// TIA Portal V17 export
// export: Created 2026-04-13T11:12:43.3625871Z, ExportSetting WithDefaults, DisplayName Totally Integrated Automation Portal, DisplayVersion V17 Update 4, DisplayName TIA Portal Openness, DisplayVersion V17 Update 4, DisplayName TIA Portal Version Control Interface, DisplayVersion V17, DisplayName SINAMICS Startdrive Advanced, DisplayVersion V17, DisplayName SINAMICS Startdrive G130, G150, S120, S150, SINAMICS MV, S210, DisplayVersion V17, DisplayName SINAMICS Startdrive G110M, G120, G120C, G120D, G120P, G115D, DisplayVersion V17, DisplayName STEP 7 Professional, DisplayVersion V17 Update 4, DisplayName STEP 7 Safety, DisplayVersion V17, DisplayName WinCC Professional, DisplayVersion V17 Update 4
FUNCTION_BLOCK "1-模拟量输出2"   // FB77, SCL
{ S7_Optimized_Access := 'TRUE' }
VERSION : 0.1
// stored: AutoNumber true, IsIECCheckEnabled false, IsRetainMemResEnabled false, MemoryReserve 100, SetENOAutomatically false, UDAEnableTagReadback false
   VAR_INPUT
      R_Max : Real;
      R_Min : Real;
      R_Value : Real;
   END_VAR
   VAR_OUTPUT
      I_ChValue : Int;
   END_VAR
BEGIN
   (**)
   #I_ChValue := REAL_TO_INT((#R_Value - #R_Min) / (#R_Max - #R_Min) * 27648.0);
END_FUNCTION_BLOCK
